FUNCTION_BLOCK FB_FeedForward_NonLinear
// LREAL: Long Real decimal number

// Input variables
VAR_INPUT
	fXDotRef 		: LREAL; // Velocity Reference [m/s]
	fMaxFlowUp 		: LREAL; // Needs to be positive (22)
	fMaxFlowDown 	: LREAL; // Needs to be positive (15)
	fDeadUp			: LREAL; // Needs to be positive (0.155)
	fDeadDown 		: LREAL; // Needs to be positive (0.18)

	fPs 			: LREAL; // [Bar]
	fPa 			: LREAL; // [Bar]
	fPb 			: LREAL; // [Bar]
	fDeltaP0		: LREAL; // [Bar]
	fAreaUp			: LREAL; // [mm^2]
	fAreaDown		: LREAL; // [mm^2]
END_VAR

// Output variables
VAR_OUTPUT
	fUFF 			: LREAL;	// FF signal value
	fFlow			: LREAL; 	// Wanted Flow
	fFlowLM			: LREAL;	// Flow [L/min]
END_VAR

// Variables
VAR
	fDeltaP_Norm	: LREAL; 	// Pressure Drop with Compensator
	
	fDeltaP			: LREAL; 	// Pressure Drop
	fDeltaP_Ref		: LREAL; 	// Reference Pressure Drop
	fFlowRef		: LREAL; 	// Reference Flow
	
	fUFFTemp		: LREAL;	// Temp Signal Out
END_VAR

// Non-linear FF compensates for disturbances where the relationship is not proportional/constant. 

fDeltaP_Norm	:= fDeltaP0 * 100000.0; // Converts from bar to Pa

IF fXDotRef > 0.0 THEN // If velocity reference > 0
	
	fFlow := fXDotRef * fAreaUp; // Calculates wanted flow 
	fFlowLM := -fFlow * 60000; // Converts flow to [L/min]. Negative sign for valve direction
	fDeltaP := (fPs - fPa) * 100000.0; // Calculates pressure drop
	IF fDeltaP < 100 THEN // Safety for pressure drop to never go below 100. Avoiding division by zero
		fDeltaP := 100;
	ELSE
		fDeltaP := fDeltaP;
	END_IF
	fDeltaP_Ref := ABS(fDeltaP_Norm/ (fDeltaP)); // Calculates reference pressure drop
	fFlowRef := (fFlow * SQRT(fDeltaP_Ref)) * 60000.0; // Calculates reference flow
	fUFFTemp := fFlowRef/fMaxFlowUp; // Normalizes output signal [0,1]
	fUFFTemp := -fUFFTemp * (1.0-fDeadUp); // Adjusts for valve deadband
	
ELSIF fXDotRef < 0.0 THEN
	
	fFlow := fXDotRef * fAreaDown;
	fFlowLM := -fFlow * 60000;
	fDeltaP := (fPs - fPb) * 100000.0;
	IF fDeltaP < 100 THEN
		fDeltaP := 100;
	ELSE
		fDeltaP := fDeltaP;
	END_IF
	fDeltaP_Ref := ABS(fDeltaP_Norm/(fDeltaP));
	fFlowRef := (fFlow * SQRT(fDeltaP_Ref)) * 60000.0;
	fUFFTemp := fFlowRef/fMaxFlowDown; 
	fUFFTemp := -fUFFTemp*(1.0-fDeadDown);
	
ELSE
	
	fUFFTemp := 0.0;		

END_IF

IF fUFFTemp > 1.0 THEN
	fUFF := 1.0;
ELSIF fUFFTemp < -1.0 THEN
	fUFF := -1.0;
ELSE
	fUFF := fUFFTemp;
END_IF

END_FUNCTION_BLOCK

(* stored: Version 1.1.0.1
   POU FB_FeedForward_NonLinear: Id {2e5cc649-f982-48da-87b8-a64d39bb47ed}, SpecialFunc None *)
